# B&R Automation Studio project A2019059_Linka_Power_CP (part 22)

#### Variables.var - Local variables
```iecst
VAR
	SC_OvlZdvihu : SequenceControlTyp;
	Zdvih_JoggDOLE : BOOL;
	Zdvih_JoggHORE : BOOL;
	Zdvih_POLOHUJ : BOOL;
	Zdvih_HOME : BOOL;
	Zdvih_STOP : BOOL;
	i : USINT;
	PrecitaneCisloPaletky : STRING[3];
	ServerOdpoved_StavPowerCP : STRING[5];
	ZadanaPoziciaUINT : UINT;
	AktualnaPoziciaUINT : UINT;
	CasPowerON : TON;
	SC_KOM_Server : SequenceControlTyp;
	Server_VyziadajStavPaletky_TYP1 : BOOL;
	Server_StavVyziadStavuPaletky : STRING[2];
	Server_PriradQRkod_TYP3 : BOOL;
	Server_StavPriradenieQRkodu : STRING[2];
	Server_VyziadajSerioveCislo_TYP0 : BOOL;
	Server_StavVyziadSeriovehoCisla : STRING[2];
	Server_OdosliStavPaletky_TYP2 : BOOL;
	Server_StavOdoslaniaStavuPaletky : STRING[2];
	Server_KomunikaciaUkoncena : BOOL;
	SKTcpClientTrace_1 : SKTcpClientTrace;
	VstupnaPremenna : STRING[80];
	VystupnaPremenna : STRING[8];
	Vysledok_OK : BOOL;
	PocetDopytovNaServer : USINT;
	CasZastaveniaServa : TON;
	TestovaciKus : BOOL;
	Revork : BOOL;
	TEST : BOOL;
	Triger_0 : BOOL;
	CisloFotky : USINT;
END_VAR
(******Zápis do ParID serva*************)
VAR
	MC_BR_ProcessParID_AcpAx_0 : MC_BR_ProcessParID_AcpAx := (0);
	McAcpAxProcessParIDType_0 : ARRAY[0..1] OF McAcpAxProcessParIDType;
	NovaHodnotaMomentu_POS : REAL := 0.0;
	NovaHodnotaMomentu_NEG : REAL := 0.0;
	PocetTrigrovKamery : USINT;
END_VAR
```

#### IOLinkKomunikacia.st
```iecst
ACTION IOLinkKomunikacia:

	//Snímač paletky//
	P1_Vytah.IN.PritomnostPaletky_S19:= P1_Vytah.PAR.SnimacPaletky_IOLinkInputs[1].0;
	P1_Vytah.IN.PrecitaneCisloPaletky_S19:= P1_Vytah.PAR.SnimacPaletky_IOLinkInputs[9];

	//Banner//
	P1_Vytah.PAR.Banner_IOLinkInputs;
	P1_Vytah.PAR.Banner_IOLinkOutputs;

	P1_Vytah.IN.BannerNalozeniaPaletky_SB11:= P1_Vytah.PAR.Banner_IOLinkInputs[1].0;

	IF P1_Vytah.OUT.Banner_CervenaLED_SB11 THEN
		P1_Vytah.PAR.Banner_IOLinkOutputs[2]:= 161;
		P1_Vytah.PAR.Banner_IOLinkOutputs[3]:= 161;
		P1_Vytah.PAR.Banner_IOLinkOutputs[4]:= 161;
		P1_Vytah.PAR.Banner_IOLinkOutputs[5]:= 161;
		P1_Vytah.PAR.Banner_IOLinkOutputs[6]:= 161;
		P1_Vytah.PAR.Banner_IOLinkOutputs[7]:= 161;
		P1_Vytah.PAR.Banner_IOLinkOutputs[8]:= 161;
		P1_Vytah.PAR.Banner_IOLinkOutputs[9]:= 161;
	ELSIF P1_Vytah.OUT.Banner_ZelenaLED_SB11 THEN
		P1_Vytah.PAR.Banner_IOLinkOutputs[2]:= 160;
		P1_Vytah.PAR.Banner_IOLinkOutputs[3]:= 160;
		P1_Vytah.PAR.Banner_IOLinkOutputs[4]:= 160;
		P1_Vytah.PAR.Banner_IOLinkOutputs[5]:= 160;
		P1_Vytah.PAR.Banner_IOLinkOutputs[6]:= 160;
		P1_Vytah.PAR.Banner_IOLinkOutputs[7]:= 160;
		P1_Vytah.PAR.Banner_IOLinkOutputs[8]:= 160;
		P1_Vytah.PAR.Banner_IOLinkOutputs[9]:= 160;
	ELSIF P1_Vytah.OUT.Banner_ModraLED_SB11 THEN
		P1_Vytah.PAR.Banner_IOLinkOutputs[2]:= 169;
		P1_Vytah.PAR.Banner_IOLinkOutputs[3]:= 169;
		P1_Vytah.PAR.Banner_IOLinkOutputs[4]:= 169;
		P1_Vytah.PAR.Banner_IOLinkOutputs[5]:= 169;
		P1_Vytah.PAR.Banner_IOLinkOutputs[6]:= 169;
		P1_Vytah.PAR.Banner_IOLinkOutputs[7]:= 169;
		P1_Vytah.PAR.Banner_IOLinkOutputs[8]:= 169;
		P1_Vytah.PAR.Banner_IOLinkOutputs[9]:= 169;
	ELSIF P1_Vytah.OUT.Banner_OranzovaLED_SB11 THEN
		P1_Vytah.PAR.Banner_IOLinkOutputs[2]:= 162;
		P1_Vytah.PAR.Banner_IOLinkOutputs[3]:= 162;
		P1_Vytah.PAR.Banner_IOLinkOutputs[4]:= 162;
		P1_Vytah.PAR.Banner_IOLinkOutputs[5]:= 162;
		P1_Vytah.PAR.Banner_IOLinkOutputs[6]:= 162;
		P1_Vytah.PAR.Banner_IOLinkOutputs[7]:= 162;
		P1_Vytah.PAR.Banner_IOLinkOutputs[8]:= 162;
		P1_Vytah.PAR.Banner_IOLinkOutputs[9]:= 162;
	ELSIF P1_Vytah.OUT.Banner_ZltaLED_SB11 THEN
		P1_Vytah.PAR.Banner_IOLinkOutputs[2]:= 164;
		P1_Vytah.PAR.Banner_IOLinkOutputs[3]:= 164;
		P1_Vytah.PAR.Banner_IOLinkOutputs[4]:= 164;
		P1_Vytah.PAR.Banner_IOLinkOutputs[5]:= 164;
		P1_Vytah.PAR.Banner_IOLinkOutputs[6]:= 164;
		P1_Vytah.PAR.Banner_IOLinkOutputs[7]:= 164;
		P1_Vytah.PAR.Banner_IOLinkOutputs[8]:= 164;
        P1_Vytah.PAR.Banner_IOLinkOutputs[9]:= 164;
    ELSIF P1_Vytah.OUT.Banner_CyanLED_SB11 THEN
        P1_Vytah.PAR.Banner_IOLinkOutputs[2]:= 167;
        P1_Vytah.PAR.Banner_IOLinkOutputs[3]:= 167;
        P1_Vytah.PAR.Banner_IOLinkOutputs[4]:= 167;
        P1_Vytah.PAR.Banner_IOLinkOutputs[5]:= 167;
        P1_Vytah.PAR.Banner_IOLinkOutputs[6]:= 167;
        P1_Vytah.PAR.Banner_IOLinkOutputs[7]:= 167;
        P1_Vytah.PAR.Banner_IOLinkOutputs[8]:= 167;
        P1_Vytah.PAR.Banner_IOLinkOutputs[9]:= 167;
     ELSIF P1_Vytah.OUT.Banner_ModraRotujucaLED_SB11 THEN
        IF EDGEPOS(Blikac200ms) THEN
            IF P1_Vytah.PAR.Banner_IOLinkOutputs[5] = 160 THEN
                P1_Vytah.PAR.Banner_IOLinkOutputs[2]:= 160;
                P1_Vytah.PAR.Banner_IOLinkOutputs[6]:= 160;
				P1_Vytah.PAR.Banner_IOLinkOutputs[3]:= 160;
				P1_Vytah.PAR.Banner_IOLinkOutputs[7]:= 160;
				P1_Vytah.PAR.Banner_IOLinkOutputs[4]:= 169;
				P1_Vytah.PAR.Banner_IOLinkOutputs[8]:= 169;
				P1_Vytah.PAR.Banner_IOLinkOutputs[5]:= 169;
				P1_Vytah.PAR.Banner_IOLinkOutputs[9]:= 169;
            ELSIF P1_Vytah.PAR.Banner_IOLinkOutputs[2] = 160 THEN
				P1_Vytah.PAR.Banner_IOLinkOutputs[2]:= 169;
				P1_Vytah.PAR.Banner_IOLinkOutputs[6]:= 169;
				P1_Vytah.PAR.Banner_IOLinkOutputs[3]:= 160;
				P1_Vytah.PAR.Banner_IOLinkOutputs[7]:= 160;
				P1_Vytah.PAR.Banner_IOLinkOutputs[4]:= 160;
				P1_Vytah.PAR.Banner_IOLinkOutputs[8]:= 160;
				P1_Vytah.PAR.Banner_IOLinkOutputs[5]:= 169;
				P1_Vytah.PAR.Banner_IOLinkOutputs[9]:= 169;
			ELSIF P1_Vytah.PAR.Banner_IOLinkOutputs[8] = 160 THEN
				P1_Vytah.PAR.Banner_IOLinkOutputs[2]:= 169;
				P1_Vytah.PAR.Banner_IOLinkOutputs[6]:= 169;
				P1_Vytah.PAR.Banner_IOLinkOutputs[3]:= 169;
				P1_Vytah.PAR.Banner_IOLinkOutputs[7]:= 169;
				P1_Vytah.PAR.Banner_IOLinkOutputs[4]:= 160;
				P1_Vytah.PAR.Banner_IOLinkOutputs[8]:= 160;
				P1_Vytah.PAR.Banner_IOLinkOutputs[5]:= 160;
				P1_Vytah.PAR.Banner_IOLinkOutputs[9]:= 160;
			ELSIF P1_Vytah.PAR.Banner_IOLinkOutputs[9] = 160 THEN
				P1_Vytah.PAR.Banner_IOLinkOutputs[2]:= 160;
				P1_Vytah.PAR.Banner_IOLinkOutputs[6]:= 160;
				P1_Vytah.PAR.Banner_IOLinkOutputs[3]:= 169;
				P1_Vytah.PAR.Banner_IOLinkOutputs[7]:= 169;
				P1_Vytah.PAR.Banner_IOLinkOutputs[4]:= 169;
				P1_Vytah.PAR.Banner_IOLinkOutputs[8]:= 169;
				P1_Vytah.PAR.Banner_IOLinkOutputs[5]:= 160;
				P1_Vytah.PAR.Banner_IOLinkOutputs[9]:= 160;
			ELSE
				P1_Vytah.PAR.Banner_IOLinkOutputs[5]:= 160;
			END_IF
		END_IF
	ELSE
		P1_Vytah.PAR.Banner_IOLinkOutputs[2]:= 0;
		P1_Vytah.PAR.Banner_IOLinkOutputs[3]:= 0;
		P1_Vytah.PAR.Banner_IOLinkOutputs[4]:= 0;
		P1_Vytah.PAR.Banner_IOLinkOutputs[5]:= 0;
		P1_Vytah.PAR.Banner_IOLinkOutputs[6]:= 0;
		P1_Vytah.PAR.Banner_IOLinkOutputs[7]:= 0;
		P1_Vytah.PAR.Banner_IOLinkOutputs[8]:= 0;
		P1_Vytah.PAR.Banner_IOLinkOutputs[9]:= 0;
	END_IF

	//Zhasnutie bannera//
	IF P1_Vytah.OUT.Banner_LED_OFF THEN
		P1_Vytah.OUT.Banner_CervenaLED_SB11:= FALSE;
		P1_Vytah.OUT.Banner_ZelenaLED_SB11:= FALSE;
		P1_Vytah.OUT.Banner_ModraLED_SB11:= FALSE;
        P1_Vytah.OUT.Banner_OranzovaLED_SB11:= FALSE;
		P1_Vytah.OUT.Banner_ModraRotujucaLED_SB11:= FALSE;
        P1_Vytah.OUT.Banner_ZltaLED_SB11:= FALSE;
        P1_Vytah.OUT.Banner_CyanLED_SB11:= FALSE;
        P1_Vytah.OUT.Banner_LED_OFF:= FALSE;
	END_IF

END_ACTION
```

#### StratoveSekundy.st
```iecst
ACTION StratoveSekundy:

END_ACTION
```

#### OvlServaZdvihu.st
```iecst
ACTION OvlServaZdvihu:

	//**************************Axis 6***********************************//
	//Otáčka serva = 5mm//
	//Motor má klasický encodér a brzdu//

    //ENABLE knižnice//
    IF P1_Vytah.ServoZdvihuVytahu_M31.STATUS.Communication_READY THEN
        P1_Vytah.ServoZdvihuVytahu_M31.CMD.ENABLE:= TRUE;
    ELSE
        P1_Vytah.ServoZdvihuVytahu_M31.CMD.ENABLE:= FALSE;
    END_IF

	//Zapnutie serva//

	CasPowerON.IN:= P1_Vytah.ServoZdvihuVytahu_M31.STATUS.ReadyToPower_ON AND P1_Vytah.STAV.ServoZvihu_LimitSnimace_BUSY AND P1_Vytah.ServoZdvihuVytahu_M31.STATUS.EnableSwitch_ACTIVE AND NOT P1_Vytah.ServoZdvihuVytahu_M31.STATUS.ERROR;
	IF CasPowerON.Q THEN
		P1_Vytah.ServoZdvihuVytahu_M31.CMD.POWER:= TRUE;
	ELSE
		P1_Vytah.ServoZdvihuVytahu_M31.CMD.POWER:= FALSE;
	END_IF

	CasPowerON.PT:= T#1s;
	CasPowerON();

	//Zobrazenie stavou a parametrov serva//
	P1_Vytah.STAV.Zdvih_AktualnaPozicia:= P1_Vytah.ServoZdvihuVytahu_M31.STATUS.ActualPosition;
	P1_Vytah.STAV.Zdvih_AktualnaRychlost:= P1_Vytah.ServoZdvihuVytahu_M31.STATUS.ActualVelocity;
	P1_Vytah.STAV.ServoZdvihu_HomingOK:= P1_Vytah.ServoZdvihuVytahu_M31.STATUS.Homing_OK;
	P1_Vytah.STAV.ServoZdvihu_BUSY:= P1_Vytah.ServoZdvihuVytahu_M31.STATUS.MoveAbsolute_BUSY;
	P1_Vytah.STAV.Zdvih_JoggLimitDosiahnuty:= P1_Vytah.ServoZdvihuVytahu_M31.STATUS.JoggLimit_Dosiahnuty;

	//Zadané parametre serva//
	P1_Vytah.ServoZdvihuVytahu_M31.HomePAR.Acceleration:= 200;
	P1_Vytah.ServoZdvihuVytahu_M31.HomePAR.HomingVelocity:= 5;
	P1_Vytah.ServoZdvihuVytahu_M31.HomePAR.StartVelocity:= 20;
	P1_Vytah.ServoZdvihuVytahu_M31.HomePAR.Position:= 0;    //Offset homing pozície pre absolutny snímač
	P1_Vytah.ServoZdvihuVytahu_M31.HomePAR.HomingMode:= 2; //0 - direct, 1- refrenčný snímač, 2 - limitný snímač, 3 - absolutny encoder, 4 - na moment//

	P1_Vytah.ServoZdvihuVytahu_M31.PAR.Acceleration:= P1_RemPremenne.P1_Vytah_RychlostZdvihu*5;
	P1_Vytah.ServoZdvihuVytahu_M31.PAR.Deceleration:= P1_RemPremenne.P1_Vytah_RychlostZdvihu*10;
	P1_Vytah.ServoZdvihuVytahu_M31.PAR.StopDeceleration:= P1_RemPremenne.P1_Vytah_RychlostZdvihu*10;
	P1_Vytah.ServoZdvihuVytahu_M31.PAR.Velocity:= P1_RemPremenne.P1_Vytah_RychlostZdvihu;
	P1_Vytah.ServoZdvihuVytahu_M31.PAR.Position:= P1_Vytah.PAR.ServoZdvihu_ZadanaPozicia;

	//Zastavenie pohybu serva//
	IF Zdvih_STOP THEN
		P1_Vytah.ServoZdvihuVytahu_M31.CMD.STOP:= TRUE;
		CasZastaveniaServa.IN:= TRUE;
		SC_OvlZdvihu.Step:= 0;
		Zdvih_STOP:= FALSE;
	END_IF

	IF CasZastaveniaServa.Q  THEN
		P1_Vytah.ServoZdvihuVytahu_M31.CMD.STOP:= FALSE;
		CasZastaveniaServa.IN:= FALSE;
	END_IF

	CasZastaveniaServa.PT:= T#2s;
	CasZastaveniaServa();

	//Prepočet pozície výťahu//
	ZadanaPoziciaUINT:= LREAL_TO_UINT(P1_Vytah.PAR.ServoZdvihu_ZadanaPozicia);
	AktualnaPoziciaUINT:= LREAL_TO_UINT(P1_Vytah.STAV.Zdvih_AktualnaPozicia);

	//Volanie funkcie SequenceControl//
	SequenceControl(SC:= SC_OvlZdvihu);

	CASE SC_OvlZdvihu.Step OF

		0:
			SC_OvlZdvihu.StepName:= '0 - Nulovanie';
			Zdvih_JoggHORE:= FALSE;
			Zdvih_JoggDOLE:= FALSE;
			Zdvih_POLOHUJ:= FALSE;
			Zdvih_HOME:= FALSE;
			P1_Vytah.ServoZdvihuVytahu_M31.CMD.HOME:= FALSE;
			P1_Vytah.ServoZdvihuVytahu_M31.CMD.JoggVPRED:= FALSE;
			P1_Vytah.ServoZdvihuVytahu_M31.CMD.JoggVZAD:= FALSE;
			P1_Vytah.ServoZdvihuVytahu_M31.CMD.MoveAbsolute:= FALSE;
            Safety.IN.P1_Vytah_Zdvih_BUSY:= FALSE;
            P1_Vytah.STAV.ServoZdvihu_Homing_BUSY:= FALSE;

			IF SC_P1_Vytah.Step <> 0 AND P1_Vytah.ServoZdvihuVytahu_M31.STATUS.Power_ON AND NOT P1_Vytah.ServoZdvihuVytahu_M31.STATUS.ERROR AND NOT P1_Vytah.ServoZdvihuVytahu_M31.STATUS.STOP_ACTIVE THEN
				SC_OvlZdvihu.ResetStep:= TRUE;
				SC_OvlZdvihu.Step:= 1;
			END_IF

		1:
			SC_OvlZdvihu.StepName:= '1 - Rozhodnutie o cinnosti';
			IF Zdvih_JoggHORE THEN
				SC_OvlZdvihu.Step:= 10;
			ELSIF Zdvih_JoggDOLE THEN
				SC_OvlZdvihu.Step:= 20;
			ELSIF Zdvih_HOME THEN
				SC_OvlZdvihu.Step:= 30;
			ELSIF Zdvih_POLOHUJ THEN
				SC_OvlZdvihu.Step:= 40;
			END_IF

		10:
			SC_OvlZdvihu.StepName:= '10 - Jogg HORE';
			SC_OvlZdvihu.IdleTime.PT:= T#3s;
			SC_OvlZdvihu.AlarmTime.PT:= T#3s;

			Safety.IN.P1_Vytah_Zdvih_BUSY:= TRUE;

			IF NOT SC_OvlZdvihu.Switch1 THEN
				P1_Vytah.ServoZdvihuVytahu_M31.CMD.JoggVPRED:= TRUE;
				SC_OvlZdvihu.Switch1:= TRUE;
			END_IF

			IF NOT Zdvih_JoggHORE THEN
				SC_OvlZdvihu.ResetStep:= TRUE;
				SC_OvlZdvihu.Step:= 0;
			END_IF

		20:
			SC_OvlZdvihu.StepName:= '20 - Jogg DOLE';
			SC_OvlZdvihu.IdleTime.PT:= T#3s;
			SC_OvlZdvihu.AlarmTime.PT:= T#3s;

			Safety.IN.P1_Vytah_Zdvih_BUSY:= TRUE;

			IF NOT SC_OvlZdvihu.Switch1 THEN
				P1_Vytah.ServoZdvihuVytahu_M31.CMD.JoggVZAD:= TRUE;
				SC_OvlZdvihu.Switch1:= TRUE;
			END_IF

			IF NOT Zdvih_JoggDOLE THEN
				SC_OvlZdvihu.ResetStep:= TRUE;
				SC_OvlZdvihu.Step:= 0;
			END_IF

		30:
			SC_OvlZdvihu.StepName:= '30 - Homing';
			SC_OvlZdvihu.IdleTime.PT:= T#500ms;
			SC_OvlZdvihu.AlarmTime.PT:= T#3s;

			Safety.IN.P1_Vytah_Zdvih_BUSY:= TRUE;
			P1_Vytah.STAV.ServoZdvihu_Homing_BUSY:= TRUE;

			IF NOT SC_OvlZdvihu.Switch1 THEN
				P1_Vytah.ServoZdvihuVytahu_M31.CMD.HOME:= TRUE;
				SC_OvlZdvihu.IdleTime.IN:= TRUE;
				SC_OvlZdvihu.Switch1:= TRUE;
			END_IF

			IF P1_Vytah.ServoZdvihuVytahu_M31.STATUS.Homing_OK AND SC_OvlZdvihu.IdleTime.Q THEN
				SC_OvlZdvihu.ResetStep:= TRUE;
				SC_OvlZdvihu.Step:= 0;
			END_IF

		40:
			SC_OvlZdvihu.StepName:= '40 - Polohovanie';
			SC_OvlZdvihu.IdleTime.PT:= T#500ms;
			SC_OvlZdvihu.AlarmTime.PT:= T#3s;

			Safety.IN.P1_Vytah_Zdvih_BUSY:= TRUE;

			IF NOT SC_OvlZdvihu.Switch1 THEN
				P1_Vytah.ServoZdvihuVytahu_M31.CMD.MoveAbsolute:= TRUE;
				SC_OvlZdvihu.Switch1:= TRUE;
			END_IF

			IF (AktualnaPoziciaUINT = ZadanaPoziciaUINT) AND P1_Vytah.ServoZdvihuVytahu_M31.STATUS.MoveAbsolute_DONE THEN
				P1_Vytah.STAV.ServoZdvihu_PoziciaDosiahnuta:= TRUE;
				SC_OvlZdvihu.ResetStep:= TRUE;
				SC_OvlZdvihu.Step:= 0;
			END_IF

	END_CASE

END_ACTION
```

### Program Logical/Program/Pracovisko_2/P2_Main (IEC)

#### Main.st - Init, cyclic, exit code
```iecst
PROGRAM _INIT
	(* Insert code here *)

END_PROGRAM

PROGRAM _CYCLIC

	//Volanie podprogramu//
    OvlVentilovychTerminalov;
    ProfinetKomunikaciaKAM1;
    ProfinetKomunikaciaKAM7;
    ProfinetKomunikaciaKAM8;
    ProfinetKomunikaciaKAM9;
    ProfinetKomunikaciaKAM10;
    ProfinetKomunikaciaKAM11;
    ProfinetKomunikaciaKAM12;
    ProfinetKomunikaciaKAM17;

    //******************************Stav moduly OK**************************************//
    IF P2_Pracovisko.STAV.ModulDI21_OK AND
        P2_Pracovisko.STAV.ModulDI22_OK AND
        P2_Pracovisko.STAV.ModulDI23_OK AND
        P2_Pracovisko.STAV.ModulDI24_OK AND
        P2_Pracovisko.STAV.ModulDI25_OK AND
        P2_Pracovisko.STAV.ModulDM21_OK AND
        P2_Pracovisko.STAV.ModulDS21_OK AND
        P2_Pracovisko.STAV.ModulDS22_OK AND
        P2_Pracovisko.STAV.ModulDS23_OK AND
        P2_Pracovisko.STAV.ModulSI21_OK AND
        P2_Pracovisko.STAV.ModulSI22_OK THEN
        P2_Pracovisko.STAV.Moduly_OK:= TRUE;
    ELSE
        P2_Pracovisko.STAV.Moduly_OK:= FALSE;
    END_IF

    //******************************Stav kamery OK**************************************//
    IF Linka.STAV.WenglorControlUnit_OK AND
        CAM8.STAV.READY AND
        CAM9.STAV.READY THEN
        P2_Pracovisko.STAV.Kamery_OK:= TRUE;
    ELSE
        P2_Pracovisko.STAV.Kamery_OK:= FALSE;
    END_IF

    //******************************Stav skrutkovačky OK*********************************//
    IF P2_Pracovisko.STAV.Skrutkovacka_M4_OK AND
        P2_Pracovisko.STAV.Skrutkovacka_M5_OK AND
        P2_Pracovisko.STAV.Skrutkovacka_M6_OK AND
        P2_Pracovisko.STAV.Maticovacka_M4_OK THEN
        P2_Pracovisko.STAV.Skrutkovacky_OK:= TRUE;
    ELSE
        P2_Pracovisko.STAV.Skrutkovacky_OK:= FALSE;
    END_IF

    //******************************Stav ventilové terminály OK***************************//
    IF P2_Pracovisko.STAV.VentilovyTerminal_VT1_OK AND
        P2_Pracovisko.STAV.VentilovyTerminal_VT2_OK AND
        P2_Pracovisko.STAV.VentilovyTerminal_VT3_OK THEN
        P2_Pracovisko.STAV.VentiloveTerminaly_OK:= TRUE;
    ELSE
        P2_Pracovisko.STAV.VentiloveTerminaly_OK:= FALSE;
    END_IF

    //Zrušenie signálu výmena gripra 4F5F//
    IF P2_Robot.KOM_OUT.ZmenaGripra_4F5F AND P2_Robot.KOM_IN.Stav_Griper4F5F_Vymeneny THEN
        P2_Robot.KOM_OUT.ZmenaGripra_4F5F:= FALSE;
    END_IF

    //Zrušenie signálu výmena gripra 5H//
    IF P2_Robot.KOM_OUT.ZmenaGripra_5H AND P2_Robot.KOM_IN.Stav_Griper5H_Vymeneny THEN
        P2_Robot.KOM_OUT.ZmenaGripra_5H:= FALSE;
    END_IF

    //Zrušenie signálu výmena gripra čistenia Power CP//
    IF P2_Robot.KOM_OUT.ZmenaGripra_Cistenie AND P2_Robot.KOM_IN.Stav_GriperCistenia_Vymeneny THEN
        P2_Robot.KOM_OUT.ZmenaGripra_Cistenie:= FALSE;
    END_IF

    //Ukončenie cyklu//
    IF P2_Pracovisko.KoniecCyklu THEN
        IF P2_Dopravniky.Automat THEN
            P2_Dopravniky.KoniecCyklu:= TRUE;
        END_IF
        IF P2_StoperZaklTesnenia.Automat THEN
            P2_StoperZaklTesnenia.KoniecCyklu:= TRUE;
        END_IF
        IF P2_ZakladacTesnenia.Automat THEN
            P2_ZakladacTesnenia.KoniecCyklu:= TRUE;
        END_IF
        IF P2_StoperMaticovacky.Automat THEN
            P2_StoperMaticovacky.KoniecCyklu:= TRUE;
        END_IF
        IF P2_StoperSrobovania.Automat THEN
            P2_StoperSrobovania.KoniecCyklu:= TRUE;
        END_IF
        IF P2_Srobovanie.Automat THEN
            P2_Srobovanie.KoniecCyklu:= TRUE;
        END_IF
        IF P2_Robot.Automat THEN
            P2_Robot.KoniecCyklu:= TRUE;
        END_IF
        IF P2_StoperZvarania.Automat THEN
            P2_StoperZvarania.KoniecCyklu:= TRUE;
        END_IF
        IF P2_Zvaranie.Automat THEN
            P2_Zvaranie.KoniecCyklu:= TRUE;
        END_IF
        IF P2_Cistenie.Automat THEN
            P2_Cistenie.KoniecCyklu:= TRUE;
        END_IF
        P2_Pracovisko.KoniecCyklu:= FALSE;
    END_IF

    //Ukončenie cyklu pri poruche//
    IF EDGEPOS(P2_PoruchaST2) THEN
        IF P2_Dopravniky.Automat THEN
            P2_Dopravniky.KoniecCyklu:= TRUE;
        END_IF
        IF P2_StoperSrobovania.Automat THEN
            P2_StoperSrobovania.KoniecCyklu:= TRUE;
        END_IF
        IF P2_Srobovanie.Automat THEN
            P2_Srobovanie.KoniecCyklu:= TRUE;
        END_IF
        IF P2_Robot.Automat THEN
            P2_Robot.KoniecCyklu:= TRUE;
        END_IF
        IF P2_StoperZvarania.Automat THEN
            P2_StoperZvarania.KoniecCyklu:= TRUE;
        END_IF
        IF P2_Zvaranie.Automat THEN
            P2_Zvaranie.KoniecCyklu:= TRUE;
        END_IF
        IF P2_Cistenie.Automat THEN
            P2_Cistenie.KoniecCyklu:= TRUE;
        END_IF

    ELSIF EDGEPOS(P2_PoruchaST3) THEN
        IF P2_Dopravniky.Automat THEN
            P2_Dopravniky.KoniecCyklu:= TRUE;
        END_IF
        IF P2_StoperMaticovacky.Automat THEN
            P2_StoperMaticovacky.KoniecCyklu:= TRUE;
        END_IF
        IF P2_Robot.Automat THEN
            P2_Robot.KoniecCyklu:= TRUE;
        END_IF
        IF P2_StoperZvarania.Automat THEN
            P2_StoperZvarania.KoniecCyklu:= TRUE;
        END_IF
        IF P2_Zvaranie.Automat THEN
            P2_Zvaranie.KoniecCyklu:= TRUE;
        END_IF
        IF P2_Cistenie.Automat THEN
            P2_Cistenie.KoniecCyklu:= TRUE;
        END_IF

    ELSIF EDGEPOS(P2_PoruchaST4) THEN
        IF P2_Dopravniky.Automat THEN
            P2_Dopravniky.KoniecCyklu:= TRUE;
        END_IF
        IF P2_StoperMaticovacky.Automat THEN
            P2_StoperMaticovacky.KoniecCyklu:= TRUE;
        END_IF
        IF P2_StoperSrobovania.Automat THEN
            P2_StoperSrobovania.KoniecCyklu:= TRUE;
        END_IF
        IF P2_Srobovanie.Automat THEN
            P2_Srobovanie.KoniecCyklu:= TRUE;
        END_IF
        IF P2_Robot.Automat THEN
            P2_Robot.KoniecCyklu:= TRUE;
        END_IF
    END_IF

    //Status prebieha ukončenie cyklu//
    IF P2_StoperZaklTesnenia.KoniecCyklu OR
        P2_ZakladacTesnenia.KoniecCyklu OR
        P2_StoperMaticovacky.KoniecCyklu OR
        P2_StoperSrobovania.KoniecCyklu OR
        P2_Srobovanie.KoniecCyklu OR
        P2_Robot.KoniecCyklu OR
        P2_StoperZvarania.KoniecCyklu OR
        P2_Zvaranie.KoniecCyklu OR
        P2_Cistenie.KoniecCyklu THEN
        P2_Pracovisko.STAV.UkoncenieCyklu_BUSY:= TRUE;
    ELSE
        P2_Pracovisko.STAV.UkoncenieCyklu_BUSY:= FALSE;
    END_IF

    //Resetovanie pracoviska po stlačení tlačítka Automat//
    IF P2_Vizu.TL_RezimAutomat THEN
        IF P2_Pracovisko.STAV.Manual THEN
            P2_Pracovisko.Reset:= TRUE;
        END_IF
        P2_Vizu.TL_RezimAutomat:= FALSE;
    END_IF

    //Resetovanie pracoviska//
    IF P2_Pracovisko.Reset THEN
        P2_Dopravniky.Reset:= TRUE;
        P2_StoperZaklTesnenia.Reset:= TRUE;
        P2_ZakladacTesnenia.Reset:= TRUE;
        P2_StoperMaticovacky.Reset:= TRUE;
        P2_StoperSrobovania.Reset:= TRUE;
        P2_Srobovanie.Reset:= TRUE;
        P2_Robot.Reset:= TRUE;
        P2_StoperZvarania.Reset:= TRUE;
        P2_Zvaranie.Reset:= TRUE;
        P2_Cistenie.Reset:= TRUE;
        P2_Pracovisko.Reset:= FALSE;
    END_IF

    //Prepnutie pracoviska do manualneho režimu//
    IF P2_Pracovisko.Manual THEN
        P2_Dopravniky.Manual:= TRUE;
        P2_StoperZaklTesnenia.Manual:= TRUE;
        P2_ZakladacTesnenia.Manual:= TRUE;
        P2_StoperMaticovacky.Manual:= TRUE;
        P2_StoperSrobovania.Manual:= TRUE;
        P2_Srobovanie.Manual:= TRUE;
        P2_Robot.Manual:= TRUE;
        P2_StoperZvarania.Manual:= TRUE;
        P2_Zvaranie.Manual:= TRUE;
        P2_Cistenie.Manual:= TRUE;
        P2_Pracovisko.Manual:= FALSE;
    END_IF

    //Spustenie pracoviska v automatickom režime//
    IF P2_Pracovisko.Automat THEN
        P2_Dopravniky.Automat:= TRUE;
        P2_StoperZaklTesnenia.Automat:= TRUE;
        P2_ZakladacTesnenia.Automat:= TRUE;
        P2_StoperMaticovacky.Automat:= TRUE;
        P2_StoperSrobovania.Automat:= TRUE;
        P2_Srobovanie.Automat:= TRUE;
        P2_Robot.Automat:= TRUE;
        P2_StoperZvarania.Automat:= TRUE;
        P2_Zvaranie.Automat:= TRUE;
        P2_Cistenie.Automat:= TRUE;
        P2_Pracovisko.Automat:= FALSE;
    END_IF

    //***************************************************Príznaky pracoviska******************************************************//
    //Príznak pracovisko stav AUTOMAT//
    IF P2_Dopravniky.Automat OR
        P2_StoperZaklTesnenia.Automat OR
        P2_ZakladacTesnenia.Automat OR
        P2_StoperMaticovacky.Automat OR
        P2_StoperSrobovania.Automat OR
        P2_Srobovanie.Automat OR
        P2_Robot.Automat OR
        P2_StoperZvarania.Automat OR
        P2_Zvaranie.Automat OR
        P2_Cistenie.Automat THEN
        P2_Pracovisko.STAV.Automat:= TRUE;
    ELSE
        P2_Pracovisko.STAV.Automat:= FALSE;
    END_IF

    //Priznak pracovisko stav MANUAL//
    IF P2_Dopravniky.Manual OR
        P2_StoperZaklTesnenia.Manual OR
        P2_ZakladacTesnenia.Manual OR
        P2_StoperMaticovacky.Manual OR
        P2_StoperSrobovania.Manual OR
        P2_Srobovanie.Manual OR
        P2_Robot.Manual OR
        P2_StoperZvarania.Manual OR
        P2_Zvaranie.Manual OR
        P2_Cistenie.Manual THEN
        P2_Pracovisko.STAV.Manual:= TRUE;
    ELSE
        P2_Pracovisko.STAV.Manual:= FALSE;
    END_IF

    //Príznak pracovisko stav PoINIT//
    IF P2_Dopravniky.STAV.PoINIT AND
        (P2_StoperZaklTesnenia.STAV.PoINIT OR NOT P2_StoperZaklTesnenia.Automat) AND
        (P2_ZakladacTesnenia.STAV.PoINIT OR NOT P2_ZakladacTesnenia.Automat) AND
        P2_Robot.STAV.PoINIT AND
        P2_StoperMaticovacky.STAV.PoINIT AND
        P2_StoperSrobovania.STAV.PoINIT AND
        P2_Srobovanie.STAV.PoINIT AND
        P2_StoperZvarania.STAV.PoINIT AND
        P2_Zvaranie.STAV.PoINIT AND
        P2_Cistenie.STAV.PoINIT THEN
        P2_Pracovisko.STAV.PoINIT:= TRUE;
    ELSE
        P2_Pracovisko.STAV.PoINIT:= FALSE;
    END_IF

    //Príznak pracovisko stav READY//
    IF SC_P2_Dopravniky.Step = 1 AND
        SC_P2_StoperZaklTesnenia.Step = 1 AND
        SC_P2_ZakladacTesnenia.Step = 1 AND
        SC_P2_StoperMaticovacky.Step = 1 AND
        SC_P2_StoperSrobovania.Step = 1 AND
        SC_P2_Srobovanie.Step = 1 AND
        SC_P2_Robot.Step = 1 AND
        SC_P2_StoperZvarania.Step = 1 AND
        SC_P2_Zvaranie.Step = 1 AND
        SC_P2_Cistenie.Step = 1	THEN
        P2_Pracovisko.STAV.READY:= TRUE;
    ELSE
        P2_Pracovisko.STAV.READY:= FALSE;
    END_IF

    //*****************************Zapnutie osvetlenia pracoviska*********************************************************//
    P2_Pracovisko.OUT.OsvetlenieBunky:= TRUE;

    P2_Pracovisko.OUT.Osvetlenie_CAM1:= TRUE;
    P2_Pracovisko.OUT.Osvetlenie_CAM7_CAM17:= TRUE;
    P2_Pracovisko.OUT.Osvetlenie_CAM10:= TRUE;
    P2_Pracovisko.OUT.Osvetlenie_CAM11:= TRUE;

    //****************************************Ovládanie majáka***********************************************//
    //Zelené svetlo//

    IF P2_Pracovisko.STAV.Automat THEN
        P2_Pracovisko.OUT.Majak_ZeleneSvetlo:= TRUE;
    ELSIF P2_Pracovisko.STAV.Manual THEN
        P2_Pracovisko.OUT.Majak_ZeleneSvetlo:= Blikac500ms;
    ELSE
        P2_Pracovisko.OUT.Majak_ZeleneSvetlo:= FALSE;
    END_IF

    //Žlté svetlo//
    IF P2_Pracovisko.STAV.Automat AND NOT P2_Pracovisko.STAV.PoINIT THEN
        P2_Pracovisko.OUT.Majak_ZlteSvetlo:= TRUE;
    ELSIF NOT P2_Robot.KOM_IN.Stav_RezimAUTOMAT THEN
        P2_Pracovisko.OUT.Majak_ZlteSvetlo:= Blikac500ms;
    ELSIF P2_Srobovanie.STAV.Zasobnik_M4_Prazdny THEN
        P2_Pracovisko.OUT.Majak_ZlteSvetlo:= Blikac500ms;
    ELSIF P2_Srobovanie.STAV.Zasobnik_M5_Prazdny THEN
        P2_Pracovisko.OUT.Majak_ZlteSvetlo:= Blikac500ms;
    ELSIF P2_Srobovanie.STAV.Zasobnik_M6_Prazdny THEN
        P2_Pracovisko.OUT.Majak_ZlteSvetlo:= Blikac500ms;
    ELSE
        P2_Pracovisko.OUT.Majak_ZlteSvetlo:= FALSE;
    END_IF

    //Červené svetlo//
    IF P2_Pracovisko.STAV.PORUCHA THEN
        P2_Pracovisko.OUT.Majak_CerveneSvetlo:= TRUE;
    ELSE
        P2_Pracovisko.OUT.Majak_CerveneSvetlo:= FALSE;
    END_IF

    //Zvuková signalizácia//
    //    IF EDGEPOS(P2_Pracovisko.STAV.PORUCHA) THEN
    //        P2_Pracovisko.OUT.Majak_Hukacka:= Blikac500ms;
    //    END_IF

    IF P2_AlarmyVizu.PotvrdAlarmy THEN
        P2_Pracovisko.OUT.Majak_Hukacka:= FALSE;
    END_IF

END_PROGRAM

PROGRAM _EXIT
	(* Insert code here *)

END_PROGRAM
```

#### OvlVentilovychTerminalov.st
```iecst
ACTION OvlVentilovychTerminalov:

	//Mapovanie ventilového terminálu - VT1//
	P2_Pracovisko.OUT.VT1_OUT1.0:= P2_StoperZaklTesnenia.OUT.ZasunStoper_YV53;
	P2_Pracovisko.OUT.VT1_OUT1.1:= P2_StoperMaticovacky.OUT.ZasunStoper_YV52;
	P2_Pracovisko.OUT.VT1_OUT1.2;
	P2_Pracovisko.OUT.VT1_OUT1.3:= P2_SkrutkovacMatic.OUT.ZasobMatic_Ofuk_RUN_YV63;
	P2_Pracovisko.OUT.VT1_OUT1.4:= P2_SkrutkovacMatic.OUT.ZasobMatic_OfukTried_RUN_YV64;
	P2_Pracovisko.OUT.VT1_OUT1.5:= P2_SkrutkovacMatic.OUT.OddelMatic_NastrelMaticu_YV65;
	P2_Pracovisko.OUT.VT1_OUT1.6;
	P2_Pracovisko.OUT.VT1_OUT1.7;

	P2_Pracovisko.OUT.VT1_OUT2.0:= P2_SkrutkovacMatic.OUT.SkrutkMatic_PrisavMatic_RUN_YV67;
	P2_Pracovisko.OUT.VT1_OUT2.1:= P2_SkrutkovacMatic.OUT.SkrutkMatic_OfukVakua_RUN_YV66;
	P2_Pracovisko.OUT.VT1_OUT2.2:= P2_SkrutkovacMatic.OUT.PosuvacMatic_PosunMaticu_YV68;
	P2_Pracovisko.OUT.VT1_OUT2.3;
	P2_Pracovisko.OUT.VT1_OUT2.4:= P2_SkrutkovacMatic.OUT.OddelMatic_PosunMaticu_YV69;
	P2_Pracovisko.OUT.VT1_OUT2.5;
	P2_Pracovisko.OUT.VT1_OUT2.6:= P2_Srobovanie.OUT.ZasobSrobM6_Ofuk_RUN_YV30;
	P2_Pracovisko.OUT.VT1_OUT2.7:= P2_Srobovanie.OUT.ZasobSrobM6_OfukTried_RUN_YV31;

	P2_Pracovisko.OUT.VT1_OUT3.0:= P2_Srobovanie.OUT.NastrelSrobM6_PosunSrobu_YV32;
	P2_Pracovisko.OUT.VT1_OUT3.1;
	P2_Pracovisko.OUT.VT1_OUT3.2:= P2_Srobovanie.OUT.NastrelSrobM6_NastrelSrobu_YV33;
	P2_Pracovisko.OUT.VT1_OUT3.3:= P2_Srobovanie.OUT.SkrutkM6_PrisavSkrutky_RUN_YV36;
	P2_Pracovisko.OUT.VT1_OUT3.4;
	P2_Pracovisko.OUT.VT1_OUT3.5:= P2_Srobovanie.OUT.SkrutkM6_OfukVakua_RUN_YV35;
	P2_Pracovisko.OUT.VT1_OUT3.6:= P2_Srobovanie.OUT.SkrutkM6_Cist_OTVOR_YV37;
	P2_Pracovisko.OUT.VT1_OUT3.7;

	P2_Pracovisko.OUT.VT1_OUT4.0:= P2_Srobovanie.OUT.SkrutkM6_Cist_Vakum_RUN_YV39;
	P2_Pracovisko.OUT.VT1_OUT4.1:= P2_Srobovanie.OUT.SkrutkM6_Cist_OfukVakua_RUN_YV38;
	P2_Pracovisko.OUT.VT1_OUT4.2:= P2_StoperSrobovania.OUT.ZasunStoper_YV56;
	P2_Pracovisko.OUT.VT1_OUT4.3:= P2_StoperZvarania.OUT.ZasunStoper_YV59;
	P2_Pracovisko.OUT.VT1_OUT4.4;
	P2_Pracovisko.OUT.VT1_OUT4.5;
	P2_Pracovisko.OUT.VT1_OUT4.6;
	P2_Pracovisko.OUT.VT1_OUT4.7;

	//Mapovanie ventilového terminálu - VT2//
	P2_Pracovisko.OUT.VT2_OUT1.0:= P2_Cistenie.OUT.VzduchPreIonizator_RUN_YV51;
	P2_Pracovisko.OUT.VT2_OUT1.1:= P2_Cistenie.OUT.Odsavanie_OfukRUN_YV50;
	P2_Pracovisko.OUT.VT2_OUT1.2:= P2_Cistenie.OUT.Odsavanie_RUN_YV49;
	P2_Pracovisko.OUT.VT2_OUT1.3:= P2_Srobovanie.OUT.ZasobSrobM4_Ofuk_RUN_YV20;
	P2_Pracovisko.OUT.VT2_OUT1.4:= P2_Srobovanie.OUT.ZasobSrobM4_OfukTried_RUN_YV21;
	P2_Pracovisko.OUT.VT2_OUT1.5:= P2_Srobovanie.OUT.NastrelSrobM4_NastrelSrobu_YV23;
	P2_Pracovisko.OUT.VT2_OUT1.6:= P2_Srobovanie.OUT.NastrelSrobM4_PosunSrobu_YV22;
	P2_Pracovisko.OUT.VT2_OUT1.7;

	P2_Pracovisko.OUT.VT2_OUT2.0:= P2_Srobovanie.OUT.SkrutkM4_PrisavSkrutky_RUN_YV26;
	P2_Pracovisko.OUT.VT2_OUT2.1:= P2_Srobovanie.OUT.SkrutkM4_OfukVakua_RUN_YV25;
	P2_Pracovisko.OUT.VT2_OUT2.2:= P2_Srobovanie.OUT.SkrutkM4_Cist_OTVOR_YV27;
	P2_Pracovisko.OUT.VT2_OUT2.3;
	P2_Pracovisko.OUT.VT2_OUT2.4:= P2_Srobovanie.OUT.SkrutkM4_Cist_OfukVakua_RUN_YV28;
	P2_Pracovisko.OUT.VT2_OUT2.5:= P2_Srobovanie.OUT.SkrutkM4_Cist_Vakum_RUN_YV29;
	P2_Pracovisko.OUT.VT2_OUT2.6:= P2_Srobovanie.OUT.ZasobSrobM5_Ofuk_RUN_YV10;
	P2_Pracovisko.OUT.VT2_OUT2.7:= P2_Srobovanie.OUT.ZasobSrobM5_OfukTried_RUN_YV11;

	P2_Pracovisko.OUT.VT2_OUT3.0:= P2_Srobovanie.OUT.NastrelSrobM5_PosunSrobu_YV12;
	P2_Pracovisko.OUT.VT2_OUT3.1;
	P2_Pracovisko.OUT.VT2_OUT3.2:= P2_Srobovanie.OUT.NastrelSrobM5_NastrelSrobu_YV13;
	P2_Pracovisko.OUT.VT2_OUT3.3:= P2_Srobovanie.OUT.SkrutkM5_PrisavSkrutky_RUN_YV16;
	P2_Pracovisko.OUT.VT2_OUT3.4:= P2_Srobovanie.OUT.SkrutkM5_OfukVakua_RUN_YV15;
	P2_Pracovisko.OUT.VT2_OUT3.5;
	P2_Pracovisko.OUT.VT2_OUT3.6:= P2_Srobovanie.OUT.SkrutkM5_Cist_OTVOR_YV19;
	P2_Pracovisko.OUT.VT2_OUT3.7;

	P2_Pracovisko.OUT.VT2_OUT4.0:= P2_Srobovanie.OUT.SkrutkM5_Cist_OfukVakua_RUN_YV17;
	P2_Pracovisko.OUT.VT2_OUT4.1:= P2_Srobovanie.OUT.SkrutkM5_Cist_Vakum_RUN_YV18;
	P2_Pracovisko.OUT.VT2_OUT4.2:= P2_Robot.OUT.OdistiGriper_YV2;
	P2_Pracovisko.OUT.VT2_OUT4.3:= P2_Robot.OUT.ZaistiGriper_YV1;
	P2_Pracovisko.OUT.VT2_OUT4.4:= P2_Robot.OUT.VypniVakum4F5F_YV7;
	P2_Pracovisko.OUT.VT2_OUT4.5:= P2_Robot.OUT.ZapniVakum4F5F_YV6;
	P2_Pracovisko.OUT.VT2_OUT4.6:= P2_Robot.OUT.VypniVakum5H_YV9;
	P2_Pracovisko.OUT.VT2_OUT4.7:= P2_Robot.OUT.ZapniVakum5H_YV8;

	//Mapovanie ventilového terminálu - VT3//
	P2_Pracovisko.OUT.VT3_OUT1.0:= P2_Zvaranie.OUT.PojazdZvarania_VLAVO_YV46;
	P2_Pracovisko.OUT.VT3_OUT1.1:= P2_Zvaranie.OUT.PojazdZvarania_VPRAVO_YV45;
	P2_Pracovisko.OUT.VT3_OUT1.2:= P2_Cistenie.OUT.Dvere_OTVOR_YV47;
	P2_Pracovisko.OUT.VT3_OUT1.3:= P2_Cistenie.OUT.Dvere_ZATVOR_YV48;
	P2_Pracovisko.OUT.VT3_OUT1.4:= P2_StoperMaticovacky.OUT.VysunCentrovanie_YV54;
	P2_Pracovisko.OUT.VT3_OUT1.5:= P2_StoperMaticovacky.OUT.ZasunCentrovanie_YV55;
	P2_Pracovisko.OUT.VT3_OUT1.6:= P2_StoperSrobovania.OUT.VysunCentrovanie_YV57;
	P2_Pracovisko.OUT.VT3_OUT1.7:= P2_StoperSrobovania.OUT.ZasunCentrovanie_YV58;

	P2_Pracovisko.OUT.VT3_OUT2.0:= P2_StoperZvarania.OUT.VysunCentrovanie_YV60;
	P2_Pracovisko.OUT.VT3_OUT2.1:= P2_StoperZvarania.OUT.ZasunCentrovanie_YV61;
	P2_Pracovisko.OUT.VT3_OUT2.2:= P2_Robot.OUT.ZatvorGriper_YV4;
	P2_Pracovisko.OUT.VT3_OUT2.3:= P2_Robot.OUT.OtvorGriper_YV3;
	P2_Pracovisko.OUT.VT3_OUT2.4;
	P2_Pracovisko.OUT.VT3_OUT2.5;
	P2_Pracovisko.OUT.VT3_OUT2.6;
	P2_Pracovisko.OUT.VT3_OUT2.7;

	P2_Pracovisko.OUT.VT3_OUT3.0:= P2_Srobovanie.OUT.SkrutkM6_VYSUN_YV34;
	P2_Pracovisko.OUT.VT3_OUT3.1;
	P2_Pracovisko.OUT.VT3_OUT3.2:= P2_Srobovanie.OUT.SkrutkM4_VYSUN_YV24;
	P2_Pracovisko.OUT.VT3_OUT3.3;
	P2_Pracovisko.OUT.VT3_OUT3.4:= P2_Srobovanie.OUT.SkrutkM5_VYSUN_YV14;
	P2_Pracovisko.OUT.VT3_OUT3.5;
	P2_Pracovisko.OUT.VT3_OUT3.6;
	P2_Pracovisko.OUT.VT3_OUT3.7;

	P2_Pracovisko.OUT.VT3_OUT4.0;
	P2_Pracovisko.OUT.VT3_OUT4.1;
	P2_Pracovisko.OUT.VT3_OUT4.2;
	P2_Pracovisko.OUT.VT3_OUT4.3;
	P2_Pracovisko.OUT.VT3_OUT4.4;
	P2_Pracovisko.OUT.VT3_OUT4.5;
	P2_Pracovisko.OUT.VT3_OUT4.6;
	P2_Pracovisko.OUT.VT3_OUT4.7;

END_ACTION
```

#### ProfinetKomunikaciaKAM1.st
```iecst
ACTION ProfinetKomunikaciaKAM1:

	//Vstupy pre kameru//
	CAM1.Profinet_PLC_OUTPUTS[0].3:= CAM1.CMD.Triger;

	//Výstupy z kamery//
	CAM1.STAV.READY:= CAM1.Profinet_PLC_INPUTS[0].0;
	CAM1.STAV.SWITCH:= CAM1.Profinet_PLC_INPUTS[0].1;
    CAM1.STAV.BUSY:= CAM1.Profinet_PLC_INPUTS[0].2;
    CAM1.STAV.Command_AKCEPTOVANY:= CAM1.Profinet_PLC_INPUTS[0].3;
    CAM1.STAV.Command_READY:= CAM1.Profinet_PLC_INPUTS[0].4;
    CAM1.STAV.Command_ERROR:= CAM1.Profinet_PLC_INPUTS[0].5;

	//Výsledky kamery//
	CAM1.RESULT.ZalozenieTesnenia_OK:= CAM1.Profinet_PLC_INPUTS[2].0;
	CAM1.RESULT.PritomnTesnenia_OK:= CAM1.Profinet_PLC_INPUTS[2].1;
	CAM1.RESULT.PritomnPowerCP_5H5F:= CAM1.Profinet_PLC_INPUTS[2].2;
	CAM1.RESULT.PritomnPowerCP_4F:= CAM1.Profinet_PLC_INPUTS[2].3;

	///Stav výsledky READY//
	IF EDGE(CAM1.STAV.SWITCH)THEN
		CAM1.STAV.Results_READY:= TRUE;
	END_IF

END_ACTION
```

#### ProfinetKomunikaciaKAM7.st
```iecst
ACTION ProfinetKomunikaciaKAM7:

	//Vstupy pre kameru//
	CAM7.Profinet_PLC_OUTPUTS[0].3:= CAM7.CMD.Triger;

	//Výstupy z kamery//
	CAM7.STAV.READY:= CAM7.Profinet_PLC_INPUTS[0].0;
	CAM7.STAV.SWITCH:= CAM7.Profinet_PLC_INPUTS[0].1;
    CAM7.STAV.BUSY:= CAM7.Profinet_PLC_INPUTS[0].2;
    CAM7.STAV.Command_AKCEPTOVANY:= CAM7.Profinet_PLC_INPUTS[0].3;
    CAM7.STAV.Command_READY:= CAM7.Profinet_PLC_INPUTS[0].4;
    CAM7.STAV.Command_ERROR:= CAM7.Profinet_PLC_INPUTS[0].5;

	//Výsledky kamery//
	CAM7.RESULT.CitanieQRkodu_Filtra5H_OK:= CAM7.Profinet_PLC_INPUTS[2].0;

	//Prečítaný QR kód fitra 5H//
	IF EDGE(CAM7.STAV.SWITCH) THEN
		brsstrcpy(ADR(CAM7.RESULT.PrecitanyQRkod_Filtra5H),ADR(CAM7.Profinet_QRkod_Znaky));
	END_IF

	//Stav výsledky READY//
	IF EDGE(CAM7.STAV.SWITCH)THEN
		CAM7.STAV.Results_READY:= TRUE;
	END_IF

END_ACTION
```

#### ProfinetKomunikaciaKAM8.st
```iecst
ACTION ProfinetKomunikaciaKAM8:

	CAM8.STAV.READY;

	//Vstupy pre kameru//
	CAM8.Profinet_PLC_OUTPUTS[0].0:= CAM8.CMD.Triger;

	//Výstupy z kamery//
	CAM8.STAV.SWITCH:= CAM8.Profinet_PLC_INPUTS[10].0;

	//Výsledky kamery//
	CAM8.RESULT.PowerCP.CitanieQRkodu_PowerCP_OK:= CAM8.Profinet_PLC_INPUTS[0].0;

	//Prečítaný QR kód DPS//
	IF EDGE(CAM8.STAV.SWITCH) THEN
		brsstrcpy(ADR(CAM8.RESULT.PowerCP.PrecitanyQRkod_PowerCP),ADR(CAM8.Profinet_QRkod_Znaky));
	END_IF

	//Stav výsledky READY//
	IF EDGE(CAM8.STAV.SWITCH)THEN
		CAM8.STAV.Results_READY:= TRUE;
	END_IF

END_ACTION
```

#### ProfinetKomunikaciaKAM9.st
```iecst
ACTION ProfinetKomunikaciaKAM9:

	CAM9.STAV.READY;

	//Vstupy pre kameru//
	CAM9.Profinet_PLC_OUTPUTS[0].0:= CAM9.CMD.Triger;

	//Výstupy z kamery//
	CAM9.STAV.SWITCH:= CAM9.Profinet_PLC_INPUTS[10].0;

	//Výsledky kamery//
	CAM9.RESULT.PowerCP.NepritomMatice:= CAM9.Profinet_PLC_INPUTS[0].0;
	CAM9.RESULT.PowerCP.PritomnBusbaru_5H:= CAM9.Profinet_PLC_INPUTS[0].1;

	//Stav výsledky READY//
	IF EDGE(CAM9.STAV.SWITCH)THEN
		CAM9.STAV.Results_READY:= TRUE;
	END_IF

END_ACTION
```

#### ProfinetKomunikaciaKAM10.st
```iecst
ACTION ProfinetKomunikaciaKAM10:

	//Vstupy pre kameru//
	CAM10.Profinet_PLC_OUTPUTS[0].3:= CAM10.CMD.Triger;

	//Výstupy z kamery//
	CAM10.STAV.READY:= CAM10.Profinet_PLC_INPUTS[0].0;
	CAM10.STAV.SWITCH:= CAM10.Profinet_PLC_INPUTS[0].1;
    CAM10.STAV.BUSY:= CAM10.Profinet_PLC_INPUTS[0].2;
    CAM10.STAV.Command_AKCEPTOVANY:= CAM10.Profinet_PLC_INPUTS[0].3;
    CAM10.STAV.Command_READY:= CAM10.Profinet_PLC_INPUTS[0].4;
    CAM10.STAV.Command_ERROR:= CAM10.Profinet_PLC_INPUTS[0].5;

	//Výsledky kamery//
	CAM10.RESULT.Paletka.Pritomn_Busbarov_5F:= CAM10.Profinet_PLC_INPUTS[2].0;
	CAM10.RESULT.Paletka.Pritomn_Busbarov_4F:= CAM10.Profinet_PLC_INPUTS[2].1;
	CAM10.RESULT.Paletka.Pritomn_Busbarov_5H:= CAM10.Profinet_PLC_INPUTS[2].2;
	CAM10.RESULT.Paletka.Pritomn_PowerCP_5H:= CAM10.Profinet_PLC_INPUTS[2].3;
	CAM10.RESULT.Paletka.Pritomn_PowerCP_4F:= CAM10.Profinet_PLC_INPUTS[2].4;
	CAM10.RESULT.Paletka.Pritomn_PowerCP_5F:= CAM10.Profinet_PLC_INPUTS[2].5;
	CAM10.RESULT.PowerCP.Pritomn_LavejSkrutkyM6_4F5F:= CAM10.Profinet_PLC_INPUTS[2].6;
	CAM10.RESULT.PowerCP.Pritomn_PravejSkrutkyM6_4F5F:= CAM10.Profinet_PLC_INPUTS[2].7;

	CAM10.RESULT.PowerCP.Pritomn_LavejM4_4F5F:= CAM10.Profinet_PLC_INPUTS[3].0;
	CAM10.RESULT.PowerCP.Pritomn_PravejM4_4F5F:= CAM10.Profinet_PLC_INPUTS[3].1;
	CAM10.RESULT.PowerCP.Pritomn_SkrutkyM4_Filtra_5H:= CAM10.Profinet_PLC_INPUTS[3].2;
	CAM10.RESULT.PowerCP.Pritomn_LavejSkrutkyM5_5H:= CAM10.Profinet_PLC_INPUTS[3].3;
	CAM10.RESULT.PowerCP.Pritomn_PravejSkrutkyM5_5H:= CAM10.Profinet_PLC_INPUTS[3].4;

	//Stav výsledky READY//
	IF EDGE(CAM10.STAV.SWITCH)THEN
		CAM10.STAV.Results_READY:= TRUE;
	END_IF

END_ACTION
```

#### ProfinetKomunikaciaKAM11.st
```iecst
ACTION ProfinetKomunikaciaKAM11:

	//Vstupy pre kameru//
	CAM11.Profinet_PLC_OUTPUTS[0].3:= CAM11.CMD.Triger;

	//Výstupy z kamery//
	CAM11.STAV.READY:= CAM11.Profinet_PLC_INPUTS[0].0;
	CAM11.STAV.SWITCH:= CAM11.Profinet_PLC_INPUTS[0].1;
    CAM11.STAV.BUSY:= CAM11.Profinet_PLC_INPUTS[0].2;
    CAM11.STAV.Command_AKCEPTOVANY:= CAM11.Profinet_PLC_INPUTS[0].3;
    CAM11.STAV.Command_READY:= CAM11.Profinet_PLC_INPUTS[0].4;
    CAM11.STAV.Command_ERROR:= CAM11.Profinet_PLC_INPUTS[0].5;

	//Výsledky kamery//
	CAM11.RESULT.PowerCP.Pritomn_PowerCP_4F:= CAM11.Profinet_PLC_INPUTS[2].0;
	CAM11.RESULT.PowerCP.Pritomn_PowerCP_5F:= CAM11.Profinet_PLC_INPUTS[2].1;
	CAM11.RESULT.PowerCP.Pritomn_PowerCP_5H:= CAM11.Profinet_PLC_INPUTS[2].2;
	CAM11.RESULT.PowerCP.Pritomn_PravyMVcase:= CAM11.Profinet_PLC_INPUTS[2].3;
	CAM11.RESULT.PowerCP.Pritomn_LavyMVcase:= CAM11.Profinet_PLC_INPUTS[2].4;
	CAM11.RESULT.PowerCP.LavyBusbar_Zvaranie_OK:= CAM11.Profinet_PLC_INPUTS[2].5;
	CAM11.RESULT.PowerCP.PravyBusbar_Zvaranie_OK:= CAM11.Profinet_PLC_INPUTS[2].6;
	CAM11.RESULT.PowerCP.Pritomn_TopCover_4F:= CAM11.Profinet_PLC_INPUTS[2].7;

	CAM11.RESULT.PowerCP.Pritomn_TopCover_5F:= CAM11.Profinet_PLC_INPUTS[3].0;
	CAM11.RESULT.PowerCP.Pritomn_TopCover_5H:= CAM11.Profinet_PLC_INPUTS[3].1;

	//Stav výsledky READY//
	IF EDGE(CAM11.STAV.SWITCH)THEN
		CAM11.STAV.Results_READY:= TRUE;
	END_IF

END_ACTION
```

#### ProfinetKomunikaciaKAM12.st
```iecst
ACTION ProfinetKomunikaciaKAM12:

	//Vstupy pre kameru//
	CAM12.Profinet_PLC_OUTPUTS[0].3:= CAM12.CMD.Triger;

	//Výstupy z kamery//
	CAM12.STAV.READY:= CAM12.Profinet_PLC_INPUTS[0].0;
	CAM12.STAV.SWITCH:= CAM12.Profinet_PLC_INPUTS[0].1;
    CAM12.STAV.BUSY:= CAM12.Profinet_PLC_INPUTS[0].2;
    CAM12.STAV.Command_AKCEPTOVANY:= CAM12.Profinet_PLC_INPUTS[0].3;
    CAM12.STAV.Command_READY:= CAM12.Profinet_PLC_INPUTS[0].4;
    CAM12.STAV.Command_ERROR:= CAM12.Profinet_PLC_INPUTS[0].5;

	//Výsledky kamery//
	CAM12.RESULT.Paletka.Pritomn_TopCover_5H5F:= CAM12.Profinet_PLC_INPUTS[2].0;
	CAM12.RESULT.Paletka.Pritomn_TopCover_4F:= CAM12.Profinet_PLC_INPUTS[2].1;
	CAM12.RESULT.Paletka.Pritomn_PravyMVcase:= CAM12.Profinet_PLC_INPUTS[2].2;
	CAM12.RESULT.Paletka.Pritomn_LavyMVcase:= CAM12.Profinet_PLC_INPUTS[2].3;

	//Stav výsledky READY//
	IF EDGE(CAM12.STAV.SWITCH)THEN
		CAM12.STAV.Results_READY:= TRUE;
	END_IF

END_ACTION
```

#### ProfinetKomunikaciaKAM17.st
```iecst
ACTION ProfinetKomunikaciaKAM17:

	//Vstupy pre kameru//
	CAM17.Profinet_PLC_OUTPUTS[0].3:= CAM17.CMD.Triger;

	//Výstupy z kamery//
	CAM17.STAV.READY:= CAM17.Profinet_PLC_INPUTS[0].0;
	CAM17.STAV.SWITCH:= CAM17.Profinet_PLC_INPUTS[0].1;
    CAM17.STAV.BUSY:= CAM17.Profinet_PLC_INPUTS[0].2;
    CAM17.STAV.Command_AKCEPTOVANY:= CAM17.Profinet_PLC_INPUTS[0].3;
    CAM17.STAV.Command_READY:= CAM17.Profinet_PLC_INPUTS[0].4;
    CAM17.STAV.Command_ERROR:= CAM17.Profinet_PLC_INPUTS[0].5;

	//Výsledky kamery//
	CAM17.RESULT.Paletka.Pritomn_TopCoveru_4F:= CAM17.Profinet_PLC_INPUTS[2].0;
	CAM17.RESULT.Paletka.Pritomn_TopCoveru_5F:= CAM17.Profinet_PLC_INPUTS[2].1;
	CAM17.RESULT.Paletka.Pritomn_TopCoveru_5H:= CAM17.Profinet_PLC_INPUTS[2].2;
	CAM17.RESULT.Paletka.Pritomn_Busbary_5H:= CAM17.Profinet_PLC_INPUTS[2].3;
	CAM17.RESULT.Paletka.Pritomn_Busbary_5F:= CAM17.Profinet_PLC_INPUTS[2].4;
	CAM17.RESULT.Paletka.Pritomn_Busbary_4F:= CAM17.Profinet_PLC_INPUTS[2].5;
	CAM17.RESULT.Paletka.Pritomn_LavyMVcase:= CAM17.Profinet_PLC_INPUTS[2].6;
	CAM17.RESULT.Paletka.Pritomn_PravyMVcase:= CAM17.Profinet_PLC_INPUTS[2].7;

	CAM17.RESULT.Paletka.Pritomn_PowerCP_4F:= CAM17.Profinet_PLC_INPUTS[3].0;
	CAM17.RESULT.Paletka.Pritomn_PowerCP_5F:= CAM17.Profinet_PLC_INPUTS[3].1;
	CAM17.RESULT.Paletka.Pritomn_PowerCP_5H:= CAM17.Profinet_PLC_INPUTS[3].2;
	CAM17.RESULT.Paletka.PoziciaBusbarov4F5F_OK:= CAM17.Profinet_PLC_INPUTS[3].4;
	CAM17.RESULT.Paletka.PoziciaBusbarov5H_OK:= CAM17.Profinet_PLC_INPUTS[3].5;

	//Stav výsledky READY//
	IF EDGE(CAM17.STAV.SWITCH)THEN
		CAM17.STAV.Results_READY:= TRUE;
	END_IF

END_ACTION
```

### Program Logical/Program/Pracovisko_2/P2_Dopravniky (IEC)

#### Main.st - Init, cyclic, exit code
```iecst
PROGRAM _INIT
	(* Insert code here *)

END_PROGRAM

PROGRAM _CYCLIC

	//Volanie funkcie SequenceControl//
	SequenceControl(SC:= SC_P2_Dopravniky);

	//Reset sekcie //
    IF NOT Safety.STAV.P2_ZonaBunky_AKTIVNA THEN
        SC_P2_Dopravniky.Step:= 0;
    ELSIF P2_Dopravniky.Reset THEN
		SC_P2_Dopravniky.Step:= 0;
		P2_Dopravniky.Reset:= FALSE;
	END_IF

	CASE SC_P2_Dopravniky.Step OF

		0:
			SC_P2_Dopravniky.StepName:='0 - Nulovanie';
			P2_Dopravniky.Automat:= FALSE;
			P2_Dopravniky.KoniecCyklu:= FALSE;
			P2_Dopravniky.Manual:= FALSE;
			P2_Dopravniky.STAV.PoINIT:= FALSE;
			P2_Dopravniky.OUT.HornyDoprav_ChodVPRED_M7:= FALSE;
			P2_Dopravniky.OUT.SpodnyDoprav_ChodVPRED_M8:= FALSE;

			IF Safety.STAV.P2_ZonaBunky_AKTIVNA AND NOT P2_Pracovisko.STAV.PORUCHA  AND P2_Pracovisko.IN.PrivodVzduchu_SnimacTlaku_S3 THEN
				SC_P2_Dopravniky.ResetStep:= TRUE;
				SC_P2_Dopravniky.Step:= 1;
			END_IF

		1:
			SC_P2_Dopravniky.StepName:='1 - Cakam na spustenie vyroby';
			P2_Dopravniky.KoniecCyklu:= FALSE;
            IF P2_Dopravniky.Automat THEN
				SC_P2_Dopravniky.Step:= 2;
			ELSIF P2_Dopravniky.Manual THEN
				SC_P2_Dopravniky.Step:= 700;
			END_IF

			//********************************************************Inicializácia****************************************************************************//

		2:
			SC_P2_Dopravniky.StepName:='2 - Inicializacia - cakam na spustenie inicializacie';
			SC_P2_Dopravniky.IdleTime.PT:= T#2s;
			SC_P2_Dopravniky.AlarmTime.PT:= T#5s;

			IF Safety.STAV.P2_ZaklTesnenia_Pojazd_ZASUNUTY AND P2_Srobovacky_VychodziaPozicia AND P2_SkrutkovacMatic.IN.SkrutkMatic_ZASUNUTY_MS9 (*AND P2_Robot.KOM_IN.Stav_RobotOdparkovany*) THEN
				SC_P2_Dopravniky.IdleTime.IN:= TRUE;
			ELSE
				SC_P2_Dopravniky.IdleTime.IN:= FALSE;
			END_IF

			IF SC_P2_Dopravniky.IdleTime.Q THEN
				SC_P2_Dopravniky.ResetStep:= TRUE;
				SC_P2_Dopravniky.Step:= 3;
			END_IF

		3:
			SC_P2_Dopravniky.StepName:='3 - Inicializacia - inicializacia stoprov';
			SC_P2_Dopravniky.IdleTime.PT:= T#1s;
			SC_P2_Dopravniky.AlarmTime.PT:= T#5s;

			IF P2_StoperMaticovacky.IN.PritomnostPaletky_S7 AND P2_StoperSrobovania.IN.PritomnostPaletky_S8 AND P2_StoperZvarania.IN.PritomnostPaletky_S9 THEN
				SC_P2_Dopravniky.ResetStep:= TRUE;
				SC_P2_Dopravniky.Step:= 5;
			ELSE
				IF NOT P2_StoperMaticovacky.IN.PritomnostPaletky_S7 THEN
					P2_StoperMaticovacky.OUT.ZasunStoper_YV52:= TRUE;
				END_IF
				IF NOT P2_StoperSrobovania.IN.PritomnostPaletky_S8 THEN
					P2_StoperSrobovania.OUT.ZasunStoper_YV56:= TRUE;
				END_IF
				IF NOT P2_StoperZvarania.IN.PritomnostPaletky_S9 THEN
					P2_StoperZvarania.OUT.ZasunStoper_YV59:= TRUE;
				END_IF
				SC_P2_Dopravniky.IdleTime.IN:= TRUE;
			END_IF

			IF SC_P2_Dopravniky.IdleTime.Q THEN
				P2_StoperMaticovacky.OUT.ZasunStoper_YV52:= FALSE;
				P2_StoperSrobovania.OUT.ZasunStoper_YV56:= FALSE;
				P2_StoperZvarania.OUT.ZasunStoper_YV59:= FALSE;
				SC_P2_Dopravniky.ResetStep:= TRUE;
				SC_P2_Dopravniky.Step:= 5;
			END_IF

		5:
			SC_P2_Dopravniky.StepName:='5 - Inicializacia - ukoncenie inicializacie';
			SC_P2_Dopravniky.IdleTime.PT:= T#4s;
			SC_P2_Dopravniky.AlarmTime.PT:= T#5s;

			P2_Dopravniky.OUT.HornyDoprav_ChodVPRED_M7:= TRUE;
			P2_Dopravniky.OUT.SpodnyDoprav_ChodVPRED_M8:= TRUE;
			SC_P2_Dopravniky.IdleTime.IN:= TRUE;

			IF SC_P2_Dopravniky.IdleTime.Q THEN
				P2_Dopravniky.STAV.PoINIT:= TRUE;
				SC_P2_Dopravniky.ResetStep:= TRUE;
				SC_P2_Dopravniky.Step:= 100;
			END_IF

		//********************************************************Automatický režim****************************************************************************//
		100:
			SC_P2_Dopravniky.StepName:='100 - Automaticky Rezim - cakam na vypnutie dopravnikou';
			SC_P2_Dopravniky.IdleTime.PT:= T#200ms;
			SC_P2_Dopravniky.AlarmTime.PT:= T#5s;

			IF P2_Dopravniky.KoniecCyklu AND NOT P2_StoperZaklTesnenia.Automat AND NOT P2_StoperMaticovacky.Automat AND NOT P2_StoperSrobovania.Automat AND NOT P2_StoperZvarania.Automat AND Safety.STAV.P3_VstupBunky_Bariera_AKTIVNA THEN
				SC_P2_Dopravniky.ResetStep:= TRUE;
				SC_P2_Dopravniky.Step:= 0;
			END_IF

			//*******************************************************Manuálny režim*******************************************************************************//
		700:
			SC_P2_Dopravniky.StepName:='700 - Manualny Rezim';
			SC_P2_Dopravniky.IdleTime.PT:= T#8s;
			SC_P2_Dopravniky.AlarmTime.PT:= T#5s;

	END_CASE

END_PROGRAM

PROGRAM _EXIT
	(* Insert code here *)

END_PROGRAM
```

### Program Logical/Program/Pracovisko_2/P2_StoperZaklTesnenia (IEC)
